// TIA Portal V21 export
TYPE "LAxisCtrl_typeGearInVelocity"
TITLE = LAxisCtrl_typeGearInVelocity
// Support: tech.team.motioncontrol@siemens.com
   STRUCT
      continuousUpdate : Bool := FALSE;   // TRUE: Specify gear ratio continuously; FALSE: Specify gear ratio once at the start of the job with a positive edge
      ratioNumerator : DInt := 1;   // Gear ratio numerator (permitted integer values: -2147483648 to 2147483647; value 0 not permitted)
      ratioDenominator : DInt := 1;   // Gear ratio denominator (permitted integer values: 1 to 2147483647)
      acceleration : LReal := -1.0;   // Acceleration for the synchronization (Value > 0.0: The specified value is used; Value = 0.0: Not permitted; Value < 0.0: The acceleration configured in "Technology object > Configuration > Extended parameters > Dynamic default values" is used. <TO>.DynamicDefaults.Acceleration)
      deceleration : LReal := -1.0;   // Deceleration for the synchronization (Value > 0.0: The specified value is used; Value = 0.0: Not permitted; Value < 0.0: The deceleration configured in "Technology object > Configuration > Extended parameters > Dynamic default values" is used. <TO>.DynamicDefaults.Deceleration)
      jerk : LReal := -1.0;   // Jerk for the synchronization (Value > 0.0: The specified value is used; Value = 0.0: No jerk limitation; Value < 0.0: The jerk configured in "Technology object > Configuration > Extended parameters > Dynamic default values" is used. <TO>.DynamicDefaults.Jerk)
      positionControlled : Bool := FALSE;   // Position control of the following axis (TRUE: Position-controlled mode; FALSE: Non-position-controlled operation)
   END_STRUCT;
END_TYPE
